PROGRAM MAIN
VAR
END_VAR

END_PROGRAM

(* stored: Version 1.1.0.1
   POU MAIN: Id {588f9257-e1cc-4736-9b8d-431f9ce101a4} *)
